(* IEC 61131-3 sources: CodesysTest/alpha/export/FBs/Fault, 7 files *)

(* ---- LogMessageType.dut.st ---- *)
(*#-#-#-#-#-#-#-#-#-#---Declaration---#-#-#-#-#-#-#-#-#-#-#-#-#*)

TYPE LogMessageType :
STRUCT
	logTime : DATE_AND_TIME;
	logMessage : STRING;
END_STRUCT
END_TYPE

(* ---- PACKAGE_TRACKING_STATE.dut.st ---- *)
(*#-#-#-#-#-#-#-#-#-#---Declaration---#-#-#-#-#-#-#-#-#-#-#-#-#*)

{attribute 'qualified_only'}
{attribute 'strict'}
TYPE PACKAGE_TRACKING_STATE :
(
	Idle := 0,
	ScanSection := 1,
	ExitSection := 2,
	TrunkSection := 3
);
END_TYPE

(* ---- PASSIVE_FAULT_TRIGGERS.dut.st ---- *)
(*#-#-#-#-#-#-#-#-#-#---Declaration---#-#-#-#-#-#-#-#-#-#-#-#-#*)

{attribute 'qualified_only'}
{attribute 'strict'}
TYPE PASSIVE_FAULT_TRIGGERS :
(
	AfterTime := 0,
	AfterTamp := 1,
	AfterSeal := 2,
	onTrunk := 3,
	AfterScanned := 4
);
END_TYPE

(* ---- FB_FaultManager.pou.st ---- *)
(*#-#-#-#-#-#-#-#-#-#---Declaration---#-#-#-#-#-#-#-#-#-#-#-#-#*)

FUNCTION_BLOCK FINAL FB_FaultManager
VAR_INPUT
	tamped : BOOL;
	sealed : BOOL;
	onTrunk : BOOL;
	ackAll : REFERENCE TO BOOL;
	collectionOfActiveFaults : REFERENCE TO FB_CollectionHandlerActiveFaults;
	collectionOfPassiveFaults : REFERENCE TO FB_CollectionHandlerPassiveFaults;
END_VAR
VAR_OUTPUT
	faultActive : BOOL;
	passiveFaultActive : BOOL;
	passiveExitConveyorOverride : BOOL;
	passiveExternalExitConveyorOverride : BOOL;
	passiveExemptFaultActive : BOOL;
	OEEExemptFaultActive : BOOL;
END_VAR
VAR
	_i, _j : INT;
	_castedFault : IFault;
	//_passiveExemptList : ARRAY [1..PASSIVE_EXEMPT_LIST_LENGTH] OF STRING := ['Pressure Bar Obstruction Detected', 'Barcode Verification Failed','Opened Bag was Removed'];
END_VAR
VAR CONSTANT
	PASSIVE_EXEMPT_LIST_LENGTH : INT := 3;

END_VAR
(*#-#-#-#-#-#-#-#-#-#---Implementation---#-#-#-#-#-#-#-#-#-#-#-#-#*)

//
//  FB_FactoryTest
//  FB/Fault/FB_FaultManager
//
//  Created by Evan Ische on 11/30/2021.
//  Copyright (C) 2021 Sharp Packaging Systems By Pregis. All rights reserved.
//

// No pointers, No good
IF NOT __ISVALIDREF(collectionOfActiveFaults) OR
   NOT __ISVALIDREF(collectionOfPassiveFaults) THEN
   RETURN;
END_IF

// Loop through passive faults checking for 'Action' completion
passiveExitConveyorOverride := FALSE;
passiveExternalExitConveyorOverride := FALSE;
FOR _i := 0 TO collectionOfPassiveFaults.totalObj DO
	IF __QUERYINTERFACE(collectionOfPassiveFaults.collection[_i], _castedFault) THEN

		// Check if active passive fault should halt the exit conveyor
		IF _castedFault.PassiveExitConeyorOverride THEN
			passiveExitConveyorOverride := TRUE;
		END_IF

		// Check if active passive fault should halt the external exit conveyor
		IF _castedFault.PassiveExternalExitConveyorOverride THEN
			passiveExternalExitConveyorOverride := TRUE;
		END_IF

		//
		CASE _castedFault.PassiveTrigger OF
			// Once Package has been tamped
			PASSIVE_FAULT_TRIGGERS.AfterTamp:
				IF tamped THEN
					_castedFault.Trigger();
				END_IF
			// Once current bag is sealed
			PASSIVE_FAULT_TRIGGERS.AfterSeal:
				IF sealed THEN
					_castedFault.Trigger();
				END_IF

			PASSIVE_FAULT_TRIGGERS.onTrunk:
				IF onTrunk THEN
					_castedFault.Trigger();
				END_IF

		END_CASE
	END_IF
END_FOR

// Ack Active & Passive Faults on reset
IF ackAll THEN
	ackAll := FALSE;
	collectionOfActiveFaults.AckAll();
	collectionOfPassiveFaults.AckAll();
END_IF

// Looks for faults matching faults in the exempt list
IF collectionOfActiveFaults.totalObj > 0 THEN

	IF collectionOfActiveFaults.totalObj = collectionOfPassiveFaults.totalObj THEN
		passiveExemptFaultActive := TRUE;
	ELSE
		passiveExemptFaultActive := FALSE;
	END_IF
END_IF

// Pass To Output
faultActive := collectionOfActiveFaults.faultActive;
passiveFaultActive := collectionOfPassiveFaults.faultPassive;

(* ---- FB_GetTime.pou.st ---- *)
(*#-#-#-#-#-#-#-#-#-#---Declaration---#-#-#-#-#-#-#-#-#-#-#-#-#*)

FUNCTION_BLOCK FB_GetTime
VAR_INPUT
END_VAR
VAR_OUTPUT
    currentDateAndTime : DATE_AND_TIME;

END_VAR
VAR
    iState                    : INT;
    udiUtcTime             : UDINT;
    udiUtcTimeLocal     : UDINT;
    strTimeDate         : SYSTIMEDATE;
    strTimeDateLocal     : SYSTIMEDATE;
    dtDateTimeUTC        : DATE_AND_TIME;
    timeLeftTime        : TIME;
    timeLeftDWORD        : DWORD;
    dDateUTC            : DATE;
    todTimeOfDayUTC        : TOD;

    tSysStartTime        : TIME;
    systimeStartNano    : SYSTIME;
    udiStartTimeResult    : UDINT;

    udiResult             : UDINT;

    GetDateAndTime            : DTU.GetDateAndTime;
    SetTimeZoneInformation    : DTU.SetTimeZoneInformation;

    dtCurrent                : DATE_AND_TIME;
    dtConcated                : DATE_AND_TIME;
    eWeekday                 : RTCLK.WEEKDAY;
    uiYear                     : UINT;
    uiMonth                     : UINT;
    uiDay                     : UINT;
    uiHour                     : UINT;
    uiMinute                 : UINT;
    uiSecond                 : UINT;

    dtuError                : DTU.ERROR;
END_VAR
(*#-#-#-#-#-#-#-#-#-#---Implementation---#-#-#-#-#-#-#-#-#-#-#-#-#*)

CASE iState OF

    0:
        iState:= 1;

    1:  // retrieves the target date and time, including the timezone information which was set before
        GetDateAndTime( xExecute:= TRUE);
        IF GetDateAndTime.xDone THEN
            dtCurrent:= GetDateAndTime.dtDateAndTime;
            GetDateAndTime(xExecute:= FALSE);
			currentDateAndTime := dtCurrent;
            //timeLeft := TIME_TO_DT(DT_TO_TIME(targetDate) - DT_TO_TIME(dttarget));
            iState:= 2;
        END_IF
        IF GetDateAndTime.xError THEN
            GetDateAndTime(xExecute:= FALSE);
            iState:= 32767;
        END_IF

    2: (*set a spedific date and time --> returns a variable of type DATE_AND_TIME
         DateConcat --> set only date information --> returns a variable of type DATE
         TODConcat  --> set only the time information  --> returns a variable of TOD (Time of day) *)
        IF dtuError = 0 THEN
            iState := 3;
        ELSE
            iState := 32767;
        END_IF

    3:  (*a DATE_AND_TIME variable is splitted in its parts, like year, month, day etc.
            DateSplit --> the same function for a DATE variable
            TODSplit  --> the same function for a TOD variable *)

        IF dtuError = 0 THEN
            iState:= 1;
        ELSE
            iState:= 32767;
        END_IF

    32767: ; //error

END_CASE

(* ---- FB_ONS.pou.st ---- *)
(*#-#-#-#-#-#-#-#-#-#---Declaration---#-#-#-#-#-#-#-#-#-#-#-#-#*)

FUNCTION_BLOCK FB_ONS
VAR_INPUT
	CLK : BOOL;
END_VAR
VAR_OUTPUT
	OSR : BOOL;
	OSF : BOOL;
END_VAR
VAR
	CLK_OSR : R_TRIG;
	CLK_OSF : F_TRIG;
END_VAR
(*#-#-#-#-#-#-#-#-#-#---Implementation---#-#-#-#-#-#-#-#-#-#-#-#-#*)

CLK_OSR(CLK := CLK, Q=> OSR);
CLK_OSF(CLK := CLK, Q=> OSF);

(* ---- FB_PackageTracker.pou.st ---- *)
(*#-#-#-#-#-#-#-#-#-#---Declaration---#-#-#-#-#-#-#-#-#-#-#-#-#*)

FUNCTION_BLOCK FB_PackageTracker
VAR_INPUT
	atExit : BOOL;
	scanned : BOOL;
	tamped : BOOL;
	enable : BOOL;
END_VAR
VAR_OUTPUT
	clear : BOOL;
END_VAR
VAR
	_state : PACKAGE_TRACKING_STATE;
	_packageAtExitTimer : Standard.TON := (PT := T#20MS);
	_packageNotAtExitTimer : Standard.TON := (PT := T#20MS);
END_VAR
(*#-#-#-#-#-#-#-#-#-#---Implementation---#-#-#-#-#-#-#-#-#-#-#-#-#*)

//
//  FB_FactoryTest
//  FB/Components/Factory Test/FB_FactoryTest
//
//  Created by Evan Ische on 12/07/2021.
//  Copyright (C) 2021 Sharp Packaging Systems By Pregis. All rights reserved.
//

//
_packageAtExitTimer(IN := atExit);
_packageNotAtExitTimer(IN := NOT _packageAtExitTimer.Q);

//
CASE _state OF
	PACKAGE_TRACKING_STATE.Idle:
		clear := FALSE;
		IF tamped THEN
			_state := PACKAGE_TRACKING_STATE.ScanSection;
		END_IF
	PACKAGE_TRACKING_STATE.ScanSection:
		IF scanned THEN
			_state := PACKAGE_TRACKING_STATE.ExitSection;
		END_IF
	PACKAGE_TRACKING_STATE.ExitSection:
		IF _packageAtExitTimer.Q THEN
			_state := PACKAGE_TRACKING_STATE.TrunkSection;
		END_IF
	PACKAGE_TRACKING_STATE.TrunkSection:
		IF _packageNotAtExitTimer.Q THEN
			clear := TRUE;
			_state := PACKAGE_TRACKING_STATE.Idle;
		END_IF
END_CASE

// Clear out state engine when no faults are present
IF NOT enable THEN
	_state :=PACKAGE_TRACKING_STATE.Idle;
END_IF
